FUNCTION_BLOCK FB_Puls_On_Off
VAR_INPUT
	bEnable		: BOOL;
	tPulsOn		: TIME:= T#5S;
	tPulsOff	: TIME:= T#5S;
END_VAR
VAR_OUTPUT
	bOut		: BOOL;
END_VAR
VAR
	tonPulsOn	: ton;
	tonPulsOff	: ton;	
END_VAR


tonPulsOn.PT:=tPulsOn;
tonPulsOn();
tonPulsOn.IN:=NOT tonPulsOff.Q AND bEnable;

tonPulsOff.PT:=tPulsOff;
tonPulsOff();
tonPulsOff.IN:=tonPulsOn.Q;

bOut:=NOT tonPulsOn.Q AND bEnable;

END_FUNCTION_BLOCK

(* stored: Version 1.1.0.1, ProductVersion 3.1.4024.11
   POU FB_Puls_On_Off: Id {0b1a6a54-debb-4d6f-9b1c-bb8895e5c483}, SpecialFunc None *)
